{attribute addProperty BoxType "KL2652-0050"}
{attribute addProperty Id "State_AutoAT %I*BOOL000State_RelayAT %I*BOOL000OutputAT %Q*BOOL000"}
{attribute addProperty CRC "3001914677"}
{attribute addProperty SizeInBites "0"}
{attribute addProperty SizeInBytes "0"}
TYPE Channel_B2ED9535 :
STRUCT
	{attribute addProperty Name "State_Auto"}
	State_Auto AT %I* : BOOL;
	{attribute addProperty Name "State_Relay"}
	State_Relay AT %I* : BOOL;
	{attribute addProperty Name "Output"}
	Output AT %Q* : BOOL;
END_STRUCT
END_TYPE

(* stored: Version 1.2.0.0, ProductVersion 3.1.4024.9
   DUT Channel_B2ED9535: Id {e057a578-8050-4fcf-8ec5-1f12b019210b} *)
